Yaskawa INFORM job: big_bent_planes_program.JBI

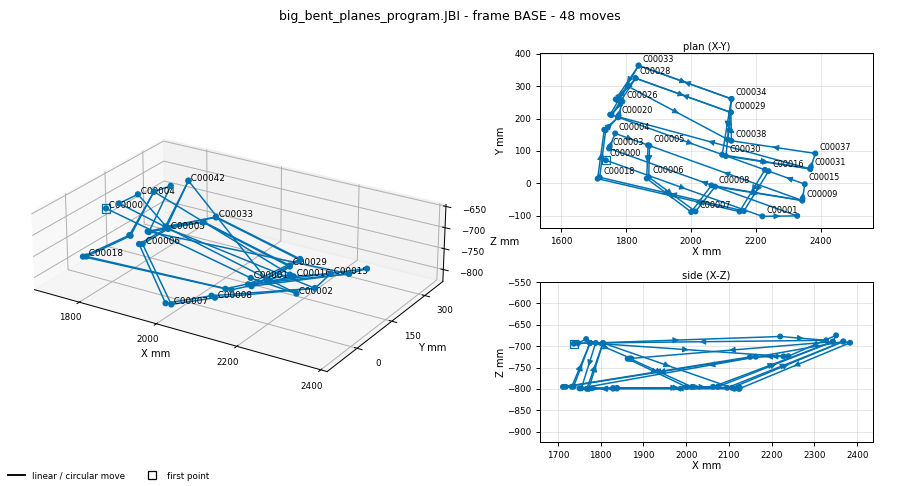
[picture p0: tool path of big_bent_planes_program.JBI in frame BASE, 48 of 50 moves have a stored position in this frame; points joined in program order, loops and branches not executed]
/JOB
//NAME big_bent_planes_program
//POS
///NPOS 48,0,48,0,0,0
///TOOL 0
///POSTYPE BASE
///RECTAN
///RCONF 0,0,0,0,0,0,0,0,0,0,0,0,0,0,0,0,0,0,0,0,0,0,0,0
C00000=1737.207623,71.314021,-693.983900,175.000000,-5.000000,5.000000
C00001=2219.856064,-101.710276,-677.206836,175.000000,-5.000000,5.000000
C00002=2327.384641,-100.240688,-686.130836,175.000000,-5.000000,5.000000
C00003=1747.161624,107.763050,-692.761836,175.000000,-5.000000,5.000000
C00004=1765.997329,154.126434,-683.216836,175.000000,-5.000000,5.000000
C00005=1871.674017,116.242473,-728.796781,175.000000,-44.714056,-19.722213
C00006=1869.461708,19.356982,-729.359017,175.000000,-44.949655,25.285224
C00007=2013.723619,-86.646592,-795.124986,-175.000000,-45.352973,115.284127
C00008=2074.213703,-10.139229,-794.873729,-175.000000,-45.285944,160.277787
C00009=2342.967076,-52.711041,-689.334836,175.000000,5.000000,5.000000
C00010=1867.419819,117.767558,-728.751671,175.000000,-44.714056,-19.722213
C00011=1863.140122,15.107998,-729.357685,175.000000,-44.948867,25.285629
C00012=2000.278528,-88.345533,-795.052615,-175.000000,-45.353886,115.283664
C00013=2062.838713,-6.061416,-794.753112,-175.000000,-45.285944,160.277787
C00014=2342.967076,-52.711041,-689.334836,175.000000,5.000000,5.000000
C00015=2350.694030,-2.365288,-674.414836,175.000000,-5.000000,5.000000
C00016=2239.004729,37.674130,-723.332930,-175.000000,-44.162920,160.277787
C00017=2162.937326,-85.333123,-724.560657,175.000000,-44.559758,115.264669
C00018=1718.157946,18.729511,-794.896203,-175.000000,-45.743219,25.287474
C00019=1736.608841,164.004282,-794.571608,175.000000,-45.837080,-19.722213
C00020=1775.253961,203.923814,-692.281836,175.000000,5.000000,5.000000
C00021=2227.639038,41.748609,-723.685827,175.000000,-44.162920,160.277787
C00022=2149.502551,-87.030266,-724.959452,175.000000,-44.559749,115.264537
C00023=1711.838617,14.480257,-795.074471,175.000000,-45.743318,25.287620
C00024=1732.358122,165.528120,-794.703590,-175.000000,-45.837080,-19.722213
C00025=1775.253961,203.923814,-692.281836,175.000000,5.000000,5.000000
C00026=1788.323959,252.354143,-692.192836,175.000000,-5.000000,5.000000
C00027=1754.770729,210.609223,-798.578160,175.000000,-45.153174,-19.722213
C00028=1828.905067,324.368284,-797.787272,175.000000,-44.956958,-64.718561
C00029=2122.446866,218.849776,-796.518287,-175.000000,-44.740030,-154.719392
C00030=2107.263306,84.244409,-797.143112,175.000000,-44.846826,160.277787
C00031=2367.546332,44.709125,-688.902836,175.000000,5.000000,5.000000
C00032=1750.517891,212.133820,-798.602316,175.000000,-45.153174,-19.722213
C00033=1838.105972,363.429439,-797.513218,175.000000,-44.956907,-64.718646
C00034=2124.528512,260.463188,-796.285420,175.000000,-44.740202,-154.719255
C00035=2095.891954,88.320917,-797.207701,175.000000,-44.846826,160.277787
C00036=2367.546332,44.709125,-688.902836,175.000000,5.000000,5.000000
C00037=2383.313518,92.268150,-691.854836,175.000000,-5.000000,5.000000
C00038=2124.426556,131.302959,-799.355235,-175.000000,-44.971303,160.277787
C00039=2122.645592,218.918466,-799.035288,175.000000,-44.827103,-154.719635
C00040=1829.010880,324.217556,-799.272518,175.000000,-44.867502,-64.717600
C00041=1771.919437,257.672987,-799.624107,-175.000000,-45.028697,-19.722213
C00042=1805.389253,299.447810,-692.469836,175.000000,5.000000,5.000000
C00043=2113.054173,135.379837,-799.367337,175.000000,-44.971303,160.277787
C00044=2124.726491,260.533735,-798.750609,175.000000,-44.827911,-154.718687
C00045=1838.209773,363.281188,-798.982375,175.000000,-44.869024,-64.717479
C00046=1767.666214,259.197721,-799.628633,175.000000,-45.028697,-19.722213
C00047=1805.389253,299.447810,-692.469836,180.000000,-60.000000,0.000000
///POSTYPE PULSE
///PULSE
EC00000=256000.0
EC00001=256000.0
EC00002=256000.0
EC00003=256000.0
EC00004=256000.0
EC00005=256000.0
EC00006=256000.0
EC00007=256000.0
EC00008=256000.0
EC00009=256000.0
EC00010=256000.0
EC00011=256000.0
EC00012=256000.0
EC00013=256000.0
EC00014=256000.0
EC00015=256000.0
EC00016=256000.0
EC00017=256000.0
EC00018=256000.0
EC00019=256000.0
EC00020=256000.0
EC00021=256000.0
EC00022=256000.0
EC00023=256000.0
EC00024=256000.0
EC00025=256000.0
EC00026=256000.0
EC00027=256000.0
EC00028=256000.0
EC00029=256000.0
EC00030=256000.0
EC00031=256000.0
EC00032=256000.0
EC00033=256000.0
EC00034=256000.0
EC00035=256000.0
EC00036=256000.0
EC00037=256000.0
EC00038=256000.0
EC00039=256000.0
EC00040=256000.0
EC00041=256000.0
EC00042=256000.0
EC00043=256000.0
EC00044=256000.0
EC00045=256000.0
EC00046=256000.0
EC00047=256000.0
//INST
///DATE 2023/08/16 12:18
///ATTR SC,RW,RJ
////FRAME BASE
///GROUP1 RB1,ST1
NOP
MOVJ P009 EX000 VJ=15.00
MOVJ C00000 EC00000 VJ=15.0
CALL JOB:SPYON
MOVL C00001 EC00001 V=150.0
MOVL C00002 EC00002 V=150.0
MOVL C00003 EC00003 V=150.0
MOVL C00004 EC00004 V=150.0
MOVL C00005 EC00005 V=150.0
MOVL C00006 EC00006 V=150.0
MOVL C00007 EC00007 V=150.0
MOVL C00008 EC00008 V=150.0
MOVL C00009 EC00009 V=150.0
MOVL C00010 EC00010 V=150.0
MOVL C00011 EC00011 V=150.0
MOVL C00012 EC00012 V=150.0
MOVL C00013 EC00013 V=150.0
MOVL C00014 EC00014 V=150.0
MOVL C00015 EC00015 V=150.0
MOVL C00016 EC00016 V=150.0
MOVL C00017 EC00017 V=150.0
MOVL C00018 EC00018 V=150.0
MOVL C00019 EC00019 V=150.0
MOVL C00020 EC00020 V=150.0
MOVL C00021 EC00021 V=150.0
MOVL C00022 EC00022 V=150.0
MOVL C00023 EC00023 V=150.0
MOVL C00024 EC00024 V=150.0
MOVL C00025 EC00025 V=150.0
MOVL C00026 EC00026 V=150.0
MOVL C00027 EC00027 V=150.0
MOVL C00028 EC00028 V=150.0
MOVL C00029 EC00029 V=150.0
MOVL C00030 EC00030 V=150.0
MOVL C00031 EC00031 V=150.0
MOVL C00032 EC00032 V=150.0
MOVL C00033 EC00033 V=150.0
MOVL C00034 EC00034 V=150.0
MOVL C00035 EC00035 V=150.0
MOVL C00036 EC00036 V=150.0
MOVL C00037 EC00037 V=150.0
MOVL C00038 EC00038 V=150.0
MOVL C00039 EC00039 V=150.0
MOVL C00040 EC00040 V=150.0
MOVL C00041 EC00041 V=150.0
MOVL C00042 EC00042 V=150.0
MOVL C00043 EC00043 V=150.0
MOVL C00044 EC00044 V=150.0
MOVL C00045 EC00045 V=150.0
MOVL C00046 EC00046 V=150.0
MOVL C00047 EC00047 V=150.0
CALL JOB:SPYOF
MOVJ P009 VJ=15.00
END
